TYPE T_FolderPath : STRING[100];
END_TYPE

(* stored: Version 1.1.0.1
   DUT T_FolderPath: Id {4e35aa58-65a1-40aa-8b91-27d2c1f16aab} *)
